{attribute 'no_explicit_call' := 'FB_EventPublisher is a CLASS and must be accessed using methods or properties'}
FUNCTION_BLOCK EventPublisherWithInheritance EXTENDS Observable IMPLEMENTS I_EventPublisher
VAR
	_event							: INT;
	eventPrev						: INT;
END_VAR


// The body of a class must not be used for code.  
// Cyclic code should be called from a method if needed.

PROPERTY PUBLIC ChangeEvent : int
SET
// IMPLEMENTED ONLY FOR TESTING PURPOSES
VAR
END_VAR
_event := changeEvent;
END_SET
END_PROPERTY

METHOD CyclicCall
IF eventPrev <> _event 			THEN
	notify();
	eventPrev := _event;
END_IF
END_METHOD

// IMPLEMENTED ONLY FOR TESTING PURPOSES
PROPERTY Event : int
GET
event := _event;
END_GET
END_PROPERTY

END_FUNCTION_BLOCK

(* stored: Version 1.1.0.1, ProductVersion 3.1.4024.11
   POU EventPublisherWithInheritance: Id {270e0f21-f10c-4d6e-aaab-748f1b75e82c}, SpecialFunc None
   Property ChangeEvent: Id {05b37224-02c8-4354-b619-b3cf8f6eb51f}
   Set Set: Id {eda01090-ae55-40a9-bf93-25e50f34c0d7}
   Method CyclicCall: Id {25dae251-2438-4d8e-9422-bfc6edc85504}
   Property Event: Id {5a53bf6d-f733-4ff7-bc62-c7e9a7ce7ec4}
   Get Get: Id {cdadf8c7-7fab-4fb4-84ee-b1e660efac40} *)
